# EPICS substitutions: iocBoot/iocsnd/snd.substitutions
file "$(TOP)/db/snd.db"{ pattern
{  BL,    DEV, GROUP,                    GAUGE}
{PINK,  SNDAL,    G1,      PINK:MAXB:S2Measure}
{PINK,  SNDAL,    G2,      PINK:MAXB:S3Measure}
{PINK,  SNDAL,    G3,      PINK:MAXA:S2Measure}
}
